FUNCTION_BLOCK Hombre EXTENDS Humano
VAR_INPUT
END_VAR
VAR_OUTPUT
END_VAR
VAR
END_VAR

END_FUNCTION_BLOCK

(* stored: Version 1.1.0.1, ProductVersion 3.1.4024.12
   POU Hombre: Id {35c1169d-1d2d-4a32-a7f1-2fe90d2d2b2c}, SpecialFunc None *)
